// TIA Portal V19 export
FUNCTION "FC20_RobotComm" : Void   // FC20, LAD
TITLE = Robot Communication
{ S7_Optimized_Access := 'TRUE' }
// stored: AutoNumber false, IsIECCheckEnabled true, SetENOAutomatically false
BEGIN

REGION Network 1: Robot communication management
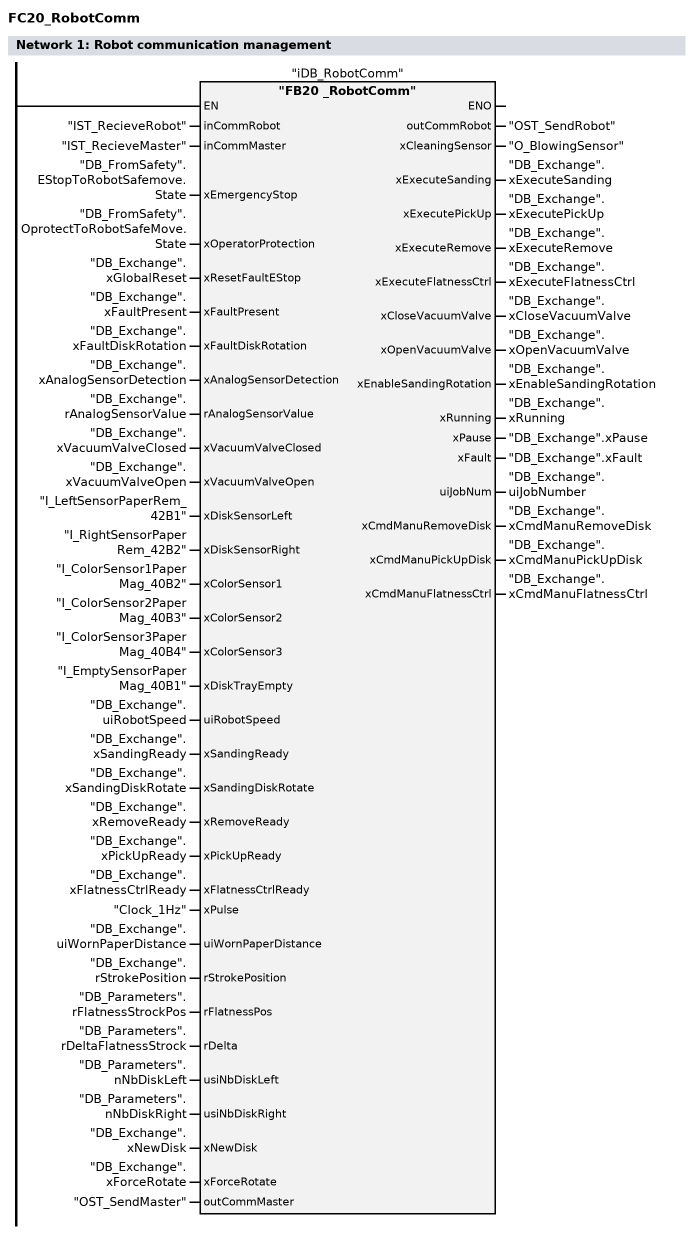
   RUNG wire#powerrail
      "iDB_RobotComm"(inCommRobot := "IST_RecieveRobot", inCommMaster := "IST_RecieveMaster", xEmergencyStop := "DB_FromSafety".EStopToRobotSafemove.State, xOperatorProtection := "DB_FromSafety".OprotectToRobotSafeMove.State, xResetFaultEStop := "DB_Exchange".xGlobalReset, xFaultPresent := "DB_Exchange".xFaultPresent, xFaultDiskRotation := "DB_Exchange".xFaultDiskRotation, xAnalogSensorDetection := "DB_Exchange".xAnalogSensorDetection, rAnalogSensorValue := "DB_Exchange".rAnalogSensorValue, xVacuumValveClosed := "DB_Exchange".xVacuumValveClosed, xVacuumValveOpen := "DB_Exchange".xVacuumValveOpen, xDiskSensorLeft := "I_LeftSensorPaperRem_42B1", xDiskSensorRight := "I_RightSensorPaperRem_42B2", xColorSensor1 := "I_ColorSensor1PaperMag_40B2", xColorSensor2 := "I_ColorSensor2PaperMag_40B3", xColorSensor3 := "I_ColorSensor3PaperMag_40B4", xDiskTrayEmpty := "I_EmptySensorPaperMag_40B1", uiRobotSpeed := "DB_Exchange".uiRobotSpeed, xSandingReady := "DB_Exchange".xSandingReady, xSandingDiskRotate := "DB_Exchange".xSandingDiskRotate, xRemoveReady := "DB_Exchange".xRemoveReady, xPickUpReady := "DB_Exchange".xPickUpReady, xFlatnessCtrlReady := "DB_Exchange".xFlatnessCtrlReady, xPulse := "Clock_1Hz", uiWornPaperDistance := "DB_Exchange".uiWornPaperDistance, rStrokePosition := "DB_Exchange".rStrokePosition, rFlatnessPos := "DB_Parameters".rFlatnessStrockPos, rDelta := "DB_Parameters".rDeltaFlatnessStrock, usiNbDiskLeft := "DB_Parameters".nNbDiskLeft, usiNbDiskRight := "DB_Parameters".nNbDiskRight, xNewDisk := "DB_Exchange".xNewDisk, xForceRotate := "DB_Exchange".xForceRotate, outCommMaster := "OST_SendMaster", outCommRobot => "OST_SendRobot", xCleaningSensor => "O_BlowingSensor", xExecuteSanding => "DB_Exchange".xExecuteSanding, xExecutePickUp => "DB_Exchange".xExecutePickUp, xExecuteRemove => "DB_Exchange".xExecuteRemove, xExecuteFlatnessCtrl => "DB_Exchange".xExecuteFlatnessCtrl, xCloseVacuumValve => "DB_Exchange".xCloseVacuumValve, xOpenVacuumValve => "DB_Exchange".xOpenVacuumValve, xEnableSandingRotation => "DB_Exchange".xEnableSandingRotation, xRunning => "DB_Exchange".xRunning, xPause => "DB_Exchange".xPause, xFault => "DB_Exchange".xFault, uiJobNum => "DB_Exchange".uiJobNumber, xCmdManuRemoveDisk => "DB_Exchange".xCmdManuRemoveDisk, xCmdManuPickUpDisk => "DB_Exchange".xCmdManuPickUpDisk, xCmdManuFlatnessCtrl => "DB_Exchange".xCmdManuFlatnessCtrl)
   END_RUNG
   // the same network as SCL:
   "iDB_RobotComm"(inCommRobot := "IST_RecieveRobot",   // "FB20 _RobotComm"
                   inCommMaster := "IST_RecieveMaster",
                   xEmergencyStop := "DB_FromSafety".EStopToRobotSafemove.State,
                   xOperatorProtection := "DB_FromSafety".OprotectToRobotSafeMove.State,
                   xResetFaultEStop := "DB_Exchange".xGlobalReset,
                   xFaultPresent := "DB_Exchange".xFaultPresent,
                   xFaultDiskRotation := "DB_Exchange".xFaultDiskRotation,
                   xAnalogSensorDetection := "DB_Exchange".xAnalogSensorDetection,
                   rAnalogSensorValue := "DB_Exchange".rAnalogSensorValue,
                   xVacuumValveClosed := "DB_Exchange".xVacuumValveClosed,
                   xVacuumValveOpen := "DB_Exchange".xVacuumValveOpen,
                   xDiskSensorLeft := "I_LeftSensorPaperRem_42B1",
                   xDiskSensorRight := "I_RightSensorPaperRem_42B2",
                   xColorSensor1 := "I_ColorSensor1PaperMag_40B2",
                   xColorSensor2 := "I_ColorSensor2PaperMag_40B3",
                   xColorSensor3 := "I_ColorSensor3PaperMag_40B4",
                   xDiskTrayEmpty := "I_EmptySensorPaperMag_40B1",
                   uiRobotSpeed := "DB_Exchange".uiRobotSpeed,
                   xSandingReady := "DB_Exchange".xSandingReady,
                   xSandingDiskRotate := "DB_Exchange".xSandingDiskRotate,
                   xRemoveReady := "DB_Exchange".xRemoveReady,
                   xPickUpReady := "DB_Exchange".xPickUpReady,
                   xFlatnessCtrlReady := "DB_Exchange".xFlatnessCtrlReady,
                   xPulse := "Clock_1Hz",
                   uiWornPaperDistance := "DB_Exchange".uiWornPaperDistance,
                   rStrokePosition := "DB_Exchange".rStrokePosition,
                   rFlatnessPos := "DB_Parameters".rFlatnessStrockPos,
                   rDelta := "DB_Parameters".rDeltaFlatnessStrock,
                   usiNbDiskLeft := "DB_Parameters".nNbDiskLeft,
                   usiNbDiskRight := "DB_Parameters".nNbDiskRight,
                   xNewDisk := "DB_Exchange".xNewDisk,
                   xForceRotate := "DB_Exchange".xForceRotate,
                   outCommMaster := "OST_SendMaster",
                   outCommRobot => "OST_SendRobot",
                   xCleaningSensor => "O_BlowingSensor",
                   xExecuteSanding => "DB_Exchange".xExecuteSanding,
                   xExecutePickUp => "DB_Exchange".xExecutePickUp,
                   xExecuteRemove => "DB_Exchange".xExecuteRemove,
                   xExecuteFlatnessCtrl => "DB_Exchange".xExecuteFlatnessCtrl,
                   xCloseVacuumValve => "DB_Exchange".xCloseVacuumValve,
                   xOpenVacuumValve => "DB_Exchange".xOpenVacuumValve,
                   xEnableSandingRotation => "DB_Exchange".xEnableSandingRotation,
                   xRunning => "DB_Exchange".xRunning,
                   xPause => "DB_Exchange".xPause,
                   xFault => "DB_Exchange".xFault,
                   uiJobNum => "DB_Exchange".uiJobNumber,
                   xCmdManuRemoveDisk => "DB_Exchange".xCmdManuRemoveDisk,
                   xCmdManuPickUpDisk => "DB_Exchange".xCmdManuPickUpDisk,
                   xCmdManuFlatnessCtrl => "DB_Exchange".xCmdManuFlatnessCtrl);
END_REGION
END_FUNCTION
